// TIA Portal V20 export
DATA_BLOCK "CallSimulation_DB"   // DB57
// stored: InstanceOfName CallSimulation, InstanceOfType FB
"CallSimulation"
   // VAR
   //    instSimRotaryAxis { ExternalAccessible := 'False'; ExternalVisible := 'False'; ExternalWritable := 'False'} : Array[0..49] of "LER_SimHmiRotaryAxis";
   //    Unwindwe1 { S7_SetPoint := 'True'} : "LER_SimHmiRotaryAxis";
   //    IEC_Timer_0_Instance { S7_SetPoint := 'True'} : TON_TIME;
   //    "LER_SimAxis+_Axis07_pnp1X" { S7_SetPoint := 'True'} : "LER_SimAxis+";
   //    "LER_SimAxis+_Axis10_pnp1Z" { S7_SetPoint := 'True'} : "LER_SimAxis+";
   //    "LER_SimAxis+_Axis8_pnp2X" { S7_SetPoint := 'True'} : "LER_SimAxis+";
   //    "LER_SimAxis+_Axis13_pnp2Z" { S7_SetPoint := 'True'} : "LER_SimAxis+";
   //    "LER_SimAxis+_Axis12_pnp1Z" { S7_SetPoint := 'True'} : "LER_SimAxis+";
   //    "LER_SimAxis+_Axis14_pnp2Z" { S7_SetPoint := 'True'} : "LER_SimAxis+";
   //    "LER_SimAxis+_Axis34_cutterX" { S7_SetPoint := 'True'} : "LER_SimAxis+";
   //    "LER_SimAxis+_Axis35_cutterZ" { S7_SetPoint := 'True'} : "LER_SimAxis+";
   //    "LER_SimAxis-_Axis36_GripperX" { S7_SetPoint := 'True'} : "LER_SimAxis-";
   //    "LER_SimAxis+_Axis37_gripperZ" { S7_SetPoint := 'True'} : "LER_SimAxis+";
   //    "LER_SimAxis-_Axis32_StackTableZ" { S7_SetPoint := 'True'} : "LER_SimAxis-";
   //    "LER_SimAxis+_Axis21_roller" { S7_SetPoint := 'True'} : "LER_SimAxis+";
   //    "LER_SimAxis+_gripperAxis_C" { S7_SetPoint := 'True'} : "LER_SimAxis+";
   //    IEC_Timer_1_Instance { S7_SetPoint := 'True'} : TON_TIME;
   //    "LER_SimAxis+_Axis05_pnp1X" { S7_SetPoint := 'True'} : "LER_SimAxis+";
   //    "LER_SimAxis+_Axis06_pnp2X" { S7_SetPoint := 'True'} : "LER_SimAxis+";
   // END_VAR
BEGIN
END_DATA_BLOCK
